Yaskawa INFORM job: TESTSRCHFFF.JBI

/JOB
//NAME TESTSRCHFFF
//POS
///NPOS 5,5,5,0,0,0
///TOOL 0
///POSTYPE PULSE
///PULSE
C00000=-135757,68735,33777,215,99269,36544
C00001=-135749,68756,34822,198,98715,36547
C00002=-135757,68506,35175,215,98292,36545
C00003=-134034,67305,33792,132,98520,37122
C00004=-132169,66242,32180,27,98966,37746
BC00000=182506,671659,131057
BC00001=182506,671659,131053
BC00002=182506,671659,131056
BC00003=182506,671659,131056
BC00004=182506,671659,131053
EC00000=798152,3
EC00001=798150,4
EC00002=798151,3
EC00003=798151,3
EC00004=798150,3
//INST
///DATE 2024/05/22 11:10
///ATTR SC,RW
///GROUP1 RB1,BS1
///GROUP2 ST1
NOP
MOVL C00000 BC00000 V=11.0  +MOVJ EC00000 VJ=0.78
SREFP 3 C00001 BC00001  +REFP EC00001
CALL JOB:SEARCH-R1-S13D
MOVL C00002 BC00002 V=11.0  +MOVJ EC00002 VJ=0.78
MOVL C00003 BC00003 V=11.0  +MOVJ EC00003 VJ=0.78
SREFP 1 C00004 BC00004  +REFP EC00004
CALL JOB:SEARCH-R1-S13DREVERSE
END
